FUNCTION_BLOCK MergeEvents (* Basic Function Block Type *)
  (* Standard: 61499-2 *)
  (* Version 0.0, 7/12/2016, Andrei, nxtControl GmbH, Template *)
  PACKAGE Main;
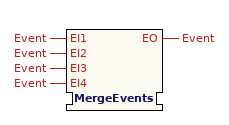
  EVENT_INPUT
    EI1; (* Normal Execution Request *)
    EI2;
    EI3;
    EI4;
  END_EVENT
  EVENT_OUTPUT
    EO; (* Execution Confirmation *)
  END_EVENT
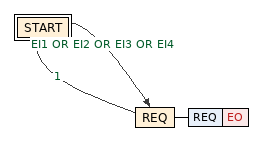
  EC_STATES
    START; (* Initial State *)
    REQ : REQ -> EO; (* Normal execution *)
  END_STATES
  EC_TRANSITIONS
    START TO REQ := EI1 OR EI2 OR EI3 OR EI4;
    REQ TO START := 1;
  END_TRANSITIONS
  ALGORITHM REQ IN ST: (* Normally executed algorithm *)
;
  END_ALGORITHM
END_FUNCTION_BLOCK
